(* CoDeSys 2.3.9.37 project: Cap5_4.pro *)
(* Libraries: Standard.lib 4.10.05 12:14:46 *)

(* Global variable list: Global_Variables *)
VAR_GLOBAL
  (* Entradas *)
  Boton : BOOL;
  BotonReset: BOOL;
  (* Salida *)
  Valor : INT;
END_VAR

(* POU PLC_PRG, ST *)
PROGRAM PLC_PRG
VAR

END_VAR

END_PROGRAM

(* Visualisation Visu
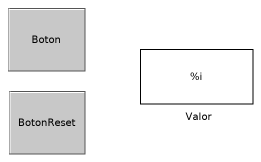
button at (30,50)-(107,113): text "Boton"; taps Boton
button at (31,133)-(107,196): text "BotonReset"; taps BotonReset
rectangle at (162,91)-(275,146): text "%i"; shows Valor
rectangle at (177,146)-(264,171): text "Valor"
*)
